// Mitsubishi GX Works2 project: 241108_PLC_STUDY3   PLC: Q02U

PROGRAM MAIN
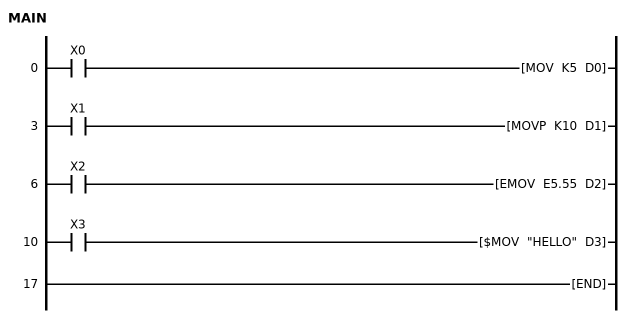
0     LD      X0
      MOV     K5 D0
3     LD      X1
      MOVP    K10 D1
6     LD      X2
      EMOV    E5.55 D2
10    LD      X3
      $MOV    "HELLO" D3
17    END
END_PROGRAM
